(* CoDeSys 2.3.9.59 project: timeStatusControl.pro *)
(* Libraries: Standard.lib, Util.lib 20.3.15 10:30:08, SysLibCallback.lib, SysLibSockets.lib, SysLibTasks.lib, SysLibRtc.lib, SysLibFile.lib, SysLibPlcCtrl.lib *)

(* POU PLC_PRG, ST *)
PROGRAM PLC_PRG
VAR
	awDateTimeDB: ARRAY [0..3] OF WORD := 4(0);		(*Data block Date and Time Galileo*)
END_VAR
awDateTimeDB;
END_PROGRAM
